// Mitsubishi GX Works2 project: 化成1TEXT01   PLC: Q03UDE

PROGRAM MAIN
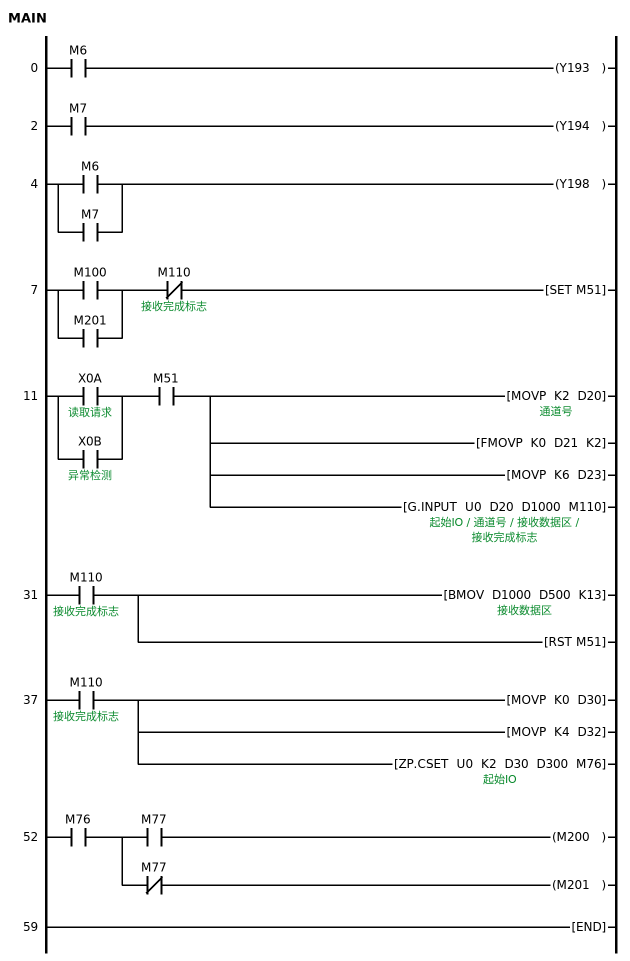
0     LD      M6
      OUT     Y193
2     LD      M7
      OUT     Y194
4     LD      M6
      OR      M7
      OUT     Y198
7     LD      M100
      OR      M201
      ANI     M110  ; 接收完成标志
      SET     M51
11    LD      X0A  ; 读取请求
      OR      X0B  ; 异常检测
      AND     M51
      MOVP    K2 D20  ; 通道号
      FMOVP   K0 D21 K2
      MOVP    K6 D23
      G.INPUT U0 D20 D1000 M110  ; 起始IO / 接收数据区
31    LD      M110  ; 接收完成标志
      BMOV    D1000 D500 K13
      RST     M51
37    LD      M110  ; 接收完成标志
      MOVP    K0 D30
      MOVP    K4 D32
      ZP.CSET U0 K2 D30 D300 M76
52    LD      M76
      MPS
      AND     M77
      OUT     M200
      MPP
      ANI     M77
      OUT     M201
59    END
END_PROGRAM
